FUNCTION_BLOCK FB_LsMdrConveyer IMPLEMENTS  I_MDRConveyer
VAR_INPUT
END_VAR
VAR_OUTPUT
END_VAR
VAR
	_Controller	: EP7402_REF;

	
END_VAR


METHOD Execute : BOOL
ADSLOGSTR(ADSLOG_MSGTYPE_LOG,'Moving Long-Straight','');
END_METHOD

PROPERTY MDRController :EP7402_REF
GET
MDRController := _Controller;
END_GET
SET
_Controller := MDRController;
END_SET
END_PROPERTY


METHOD Reset : BOOL
ADSLOGSTR(ADSLOG_MSGTYPE_LOG,'Reseting Long-straight','');
END_METHOD


METHOD Start : BOOL
ADSLOGSTR(ADSLOG_MSGTYPE_LOG,'Powering on Long-straight','');
END_METHOD


METHOD Stop : BOOL
ADSLOGSTR(ADSLOG_MSGTYPE_LOG,'Stopping Long-straight','');
END_METHOD

END_FUNCTION_BLOCK

(* stored: Version 1.1.0.1, ProductVersion 3.1.4024.6
   POU FB_LsMdrConveyer: Id {40d5586d-c049-4691-baf3-cfef919e32b3}, SpecialFunc None
   Method Execute: Id {c7952c4b-b210-44b3-aaa7-8e2c9bc33372}
   Property MDRController: Id {fefea5c4-79e4-47cf-a57a-3b3028e1c716}
   Get Get: Id {11209dd0-c62d-4ebf-91a8-ae227a07d531}
   Set Set: Id {d7c3e5e6-5411-4a02-94bb-427557a523f7}
   Method Reset: Id {fd0699e1-eccb-4e04-9ea7-0e2afc58ca01}
   Method Start: Id {f55e6142-613e-477b-83b2-2334085c1efd}
   Method Stop: Id {c9c74106-12fb-4431-955f-d91d3e05290b} *)
